{attribute 'qualified_only'}
{attribute 'strict'}
{attribute 'to_string'}
TYPE EFoerderband :
(
	Off:=0,
	init := 1,
	ErrorState := 99,
	Resolve := 100,
	Ready := 2,
	CNV_on := 3,
	CNV:aus := 4,
	Done := 5
	
);
END_TYPE

(* stored: Version 1.1.0.1
   DUT EFoerderband: Id {febd0df0-1fd4-4009-9c68-79c2893b4396} *)
